TYPE E_NeedlePoint :
STRUCT
	default				:0,
	AllocateLeft 		:1,
	AllocateRight 		:2,
	TurntableLeft       :3,
	TurntableRight		:4,
END_STRUCT
END_TYPE

(* stored: Version 1.1.0.1, ProductVersion 3.1.4024.13
   DUT E_NeedlePoint: Id {08d36390-6904-4a13-9b2b-0df3aa5376a9} *)
